FUNCTION_BLOCK FB_SiliconeProcess
VAR
    eState                  : E_SiliconeProcessState := E_SiliconeProcessState.Idle;
    bStartRequest           : BOOL;
    bStopRequest            : BOOL;
    bResetRequest           : BOOL;
    bReady                  : BOOL;
    bBusy                   : BOOL;
    bDone                   : BOOL;
    bFaulted                : BOOL;
	
	bVacuumBuildTimeoutFault   : BOOL;
	bVacuumLostFault           : BOOL;
	bVacuumReleaseTimeoutFault : BOOL;
	bEquipmentCompleteTimeoutFault : BOOL;

	
    bPinchValveRequest      : BOOL;
    bEquipmentStartRequest  : BOOL;
    bEquipmentStopRequest   : BOOL;
    bEquipmentResetRequest  : BOOL;
    stResult                : ST_ProcessResult;
    tonStep                 : TON;
	tSiliconeAirDelay 		: TIME;
END_VAR

// Runtime behaviour is implemented in Cyclic().

METHOD PUBLIC Cyclic
VAR_INPUT
    bSupplyReady               : BOOL;
    bEquipmentReady            : BOOL;
    bEquipmentBusy             : BOOL;
    bEquipmentDone             : BOOL;
    bEquipmentFaulted          : BOOL;
    stEquipmentResult          : ST_ProcessResult;
	bSiliconeStationPartPresent : BOOL;

    bSiliconeSupportExtended   : BOOL;
    bExtractorReady            : BOOL;
    bPartVacuumOk              : BOOL;
	tPartVacuumBuildTimeout    : TIME;
	tPartVacuumReleaseTimeout  : TIME;


    tPinchSettlingDelay        : TIME;
    tEquipmentStartTimeout     : TIME;
    tEquipmentCompleteTimeout  : TIME;
END_VAR

VAR_OUTPUT
    bPartVacuumEnable          : BOOL;
    bSiliconeAirEnable         : BOOL;
END_VAR
// Default one-scan handshake outputs.
bEquipmentStartRequest := FALSE;
bEquipmentStopRequest := FALSE;
bEquipmentResetRequest := FALSE;
bPartVacuumEnable := FALSE;
bSiliconeAirEnable := FALSE;

// Stop/reset are handled before state logic.
IF bResetRequest THEN
    bResetRequest := FALSE;
    bStartRequest := FALSE;
    bStopRequest := FALSE;
    bPinchValveRequest := FALSE;
    bPartVacuumEnable := FALSE;
	bSiliconeAirEnable := FALSE;
    bReady := bSupplyReady AND bEquipmentReady AND NOT bEquipmentFaulted;
    bBusy := FALSE;
    bDone := FALSE;
    bFaulted := FALSE;
	bVacuumBuildTimeoutFault := FALSE;
	bVacuumLostFault := FALSE;
	bVacuumReleaseTimeoutFault := FALSE;
	bEquipmentCompleteTimeoutFault := FALSE;
    stResult.bValid := FALSE;
    stResult.bPassed := FALSE;
    stResult.eCode := E_ProcessResultCode.None;
    stResult.udiFaultCode := 0;
    stResult.udiAlertCode := 0;
    stResult.usiRecipe := 0;
    bEquipmentResetRequest := TRUE;
    eState := E_SiliconeProcessState.Idle;
    tonStep(IN := FALSE);
    RETURN;
END_IF

IF bStopRequest THEN
    bStopRequest := FALSE;
    bStartRequest := FALSE;
    bPinchValveRequest := FALSE;
    bPartVacuumEnable := FALSE;
	bSiliconeAirEnable := FALSE;
    bBusy := FALSE;
    bDone := FALSE;
    bEquipmentStopRequest := TRUE;
    eState := E_SiliconeProcessState.Idle;
    tonStep(IN := FALSE);
    RETURN;
END_IF

// Any equipment fault while processing closes the flow path immediately.
IF bEquipmentFaulted
    AND (eState <> E_SiliconeProcessState.Idle)
    AND (eState <> E_SiliconeProcessState.Complete)
    AND (eState <> E_SiliconeProcessState.Fault)
THEN

    bPinchValveRequest := FALSE;
    bPartVacuumEnable := FALSE;
	bSiliconeAirEnable := FALSE;
    bBusy := FALSE;
    bDone := FALSE;
    bReady := FALSE;
    bFaulted := TRUE;

    stResult.bValid := FALSE;
    stResult.bPassed := FALSE;
    stResult.eCode := E_ProcessResultCode.EquipmentFault;

    eState := E_SiliconeProcessState.Fault;
END_IF

// Part holding vacuum must remain established while
// the silicone process is active.
IF NOT bPartVacuumOk
    AND (
        eState = E_SiliconeProcessState.WaitingAirBeforeSilicone
        OR eState = E_SiliconeProcessState.OpeningPinchValve
        OR eState = E_SiliconeProcessState.WaitingPinchSettling
        OR eState = E_SiliconeProcessState.StartingEquipment
        OR eState = E_SiliconeProcessState.WaitingEquipmentBusy
        OR eState = E_SiliconeProcessState.WaitingEquipmentComplete
        OR eState = E_SiliconeProcessState.ClosingPinchValve
        OR eState = E_SiliconeProcessState.WaitingAirAfterSilicone
    )
THEN

    bPinchValveRequest 			:= FALSE;
    bPartVacuumEnable 			:= FALSE;
	bSiliconeAirEnable 			:= FALSE;

    bEquipmentStartRequest 		:= FALSE;
    bEquipmentStopRequest 		:= TRUE;
	bVacuumLostFault 			:= TRUE;

    bReady 						:= FALSE;
    bBusy 						:= FALSE;
    bDone 						:= FALSE;
    bFaulted 					:= TRUE;
	stResult.bValid 			:= FALSE;
	stResult.bPassed 			:= FALSE;

    tonStep(IN := FALSE);
    eState 						:= E_SiliconeProcessState.Fault;

END_IF


CASE eState OF

    E_SiliconeProcessState.Idle:

        tonStep(IN := FALSE);

        bPinchValveRequest := FALSE;
        bPartVacuumEnable := FALSE;
		bSiliconeAirEnable := FALSE;
        bBusy := FALSE;
        bDone := FALSE;

        bReady :=
            bSupplyReady
            AND bEquipmentReady
            AND bSiliconeSupportExtended
            AND bExtractorReady
            AND NOT bEquipmentFaulted;

        IF bStartRequest AND bReady THEN
            bStartRequest := FALSE;
            bReady := FALSE;
            bBusy := TRUE;

            stResult.bValid := FALSE;
            stResult.bPassed := FALSE;

            eState := E_SiliconeProcessState.StartingVacuum;
        END_IF


   	E_SiliconeProcessState.StartingVacuum:

			bPinchValveRequest := FALSE;
			tonStep(IN := FALSE);
		
			// The part can only be detected after the Silicone Support is extended.
			// If no part is detected, finish the Silicone process as a valid FAIL.
			// Do not start the vacuum and do not run the IVEK.
			IF NOT bSiliconeStationPartPresent THEN
		
				bPartVacuumEnable := FALSE;
		
				bBusy := FALSE;
				bDone := TRUE;
				bReady := FALSE;
				bFaulted := FALSE;
		
				stResult.bValid := TRUE;
				stResult.bPassed := FALSE;
				stResult.eCode := E_ProcessResultCode.Fail;
		
				eState := E_SiliconeProcessState.Complete;
		
			ELSE
		
				bPartVacuumEnable := TRUE;
		
				eState := E_SiliconeProcessState.WaitingVacuumReady;
		
			END_IF
	
	
	E_SiliconeProcessState.WaitingVacuumReady:
	
		bPartVacuumEnable := TRUE;
		bPinchValveRequest := FALSE;
	
		tonStep(
			IN := TRUE,
			PT := tPartVacuumBuildTimeout
		);
	
		IF bPartVacuumOk THEN

			tonStep(IN := FALSE);
		
			eState := E_SiliconeProcessState.WaitingAirBeforeSilicone;
	
		ELSIF tonStep.Q THEN
	
			bPartVacuumEnable := FALSE;
			bPinchValveRequest := FALSE;
	
			bVacuumBuildTimeoutFault := TRUE;
			bFaulted := TRUE;
			bBusy := FALSE;
			bReady := FALSE;
			bDone := FALSE;
			
			stResult.bValid := FALSE;
			stResult.bPassed := FALSE;
	
			tonStep(IN := FALSE);
	
			eState := E_SiliconeProcessState.Fault;
	
		END_IF
		
		
	E_SiliconeProcessState.WaitingAirBeforeSilicone:

			bPartVacuumEnable := TRUE;
			bPinchValveRequest := FALSE;
			bSiliconeAirEnable := TRUE;
		
			tonStep(
				IN := TRUE,
				PT := tSiliconeAirDelay
			);
		
			IF tonStep.Q THEN
		
				tonStep(IN := FALSE);
		
				eState := E_SiliconeProcessState.OpeningPinchValve;
		
			END_IF
		
    E_SiliconeProcessState.OpeningPinchValve:

        bPartVacuumEnable := TRUE;
        bPinchValveRequest := TRUE;
		bSiliconeAirEnable := TRUE;

        tonStep(IN := FALSE);

        eState := E_SiliconeProcessState.WaitingPinchSettling;


    E_SiliconeProcessState.WaitingPinchSettling:

        bPartVacuumEnable := TRUE;
        bPinchValveRequest := TRUE;
		bSiliconeAirEnable := TRUE;

        tonStep(
            IN := TRUE,
            PT := tPinchSettlingDelay
        );

        IF tonStep.Q THEN
            tonStep(IN := FALSE);
            eState := E_SiliconeProcessState.StartingEquipment;
        END_IF


    E_SiliconeProcessState.StartingEquipment:

        bPartVacuumEnable := TRUE;
        bPinchValveRequest := TRUE;
		bSiliconeAirEnable := TRUE;

        IF bEquipmentReady THEN
            bEquipmentStartRequest := TRUE;

            tonStep(IN := FALSE);

            eState := E_SiliconeProcessState.WaitingEquipmentBusy;

        ELSE

            tonStep(
                IN := TRUE,
                PT := tEquipmentStartTimeout
            );

            IF tonStep.Q THEN
                bPinchValveRequest := FALSE;
                bPartVacuumEnable := FALSE;
				bSiliconeAirEnable := FALSE;
                bFaulted := TRUE;
                bBusy := FALSE;
				stResult.bValid := FALSE;
				stResult.bPassed := FALSE;

                eState := E_SiliconeProcessState.Fault;
            END_IF

        END_IF


    E_SiliconeProcessState.WaitingEquipmentBusy:

        bPartVacuumEnable := TRUE;
        bPinchValveRequest := TRUE;
		bSiliconeAirEnable := TRUE;

        // Keep Start asserted until the equipment acknowledges
        // the command by becoming Busy or Done.
        bEquipmentStartRequest := TRUE;

        tonStep(
            IN := TRUE,
            PT := tEquipmentStartTimeout
        );

        IF bEquipmentBusy OR bEquipmentDone THEN

            bEquipmentStartRequest := FALSE;

            tonStep(IN := FALSE);

            eState :=
                E_SiliconeProcessState.WaitingEquipmentComplete;

        ELSIF tonStep.Q THEN

            bEquipmentStartRequest := FALSE;
            bPinchValveRequest := FALSE;
            bPartVacuumEnable := FALSE;
			bSiliconeAirEnable := FALSE;
            bEquipmentStopRequest := TRUE;

            bFaulted := TRUE;
            bBusy := FALSE;
			stResult.bValid := FALSE;
			stResult.bPassed := FALSE;

            eState := E_SiliconeProcessState.Fault;

        END_IF


    E_SiliconeProcessState.WaitingEquipmentComplete:

        bPartVacuumEnable := TRUE;
        bPinchValveRequest := TRUE;
		bSiliconeAirEnable := TRUE;
		//bEquipmentCompleteTimeoutFault := TRUE;

        tonStep(
            IN := TRUE,
            PT := tEquipmentCompleteTimeout
        );

        IF bEquipmentDone THEN

            tonStep(IN := FALSE);
            eState := E_SiliconeProcessState.ClosingPinchValve;

        ELSIF tonStep.Q THEN

			bPinchValveRequest := FALSE;
			bPartVacuumEnable := FALSE;
			bSiliconeAirEnable := FALSE;
			bEquipmentStopRequest := TRUE;
		
			bEquipmentCompleteTimeoutFault := TRUE;
		
			bFaulted := TRUE;
			bBusy := FALSE;
		
			stResult.bValid := FALSE;
			stResult.bPassed := FALSE;
		
			eState := E_SiliconeProcessState.Fault;
		
		END_IF


    E_SiliconeProcessState.ClosingPinchValve:

			bPartVacuumEnable := TRUE;
			bSiliconeAirEnable := TRUE;
			bPinchValveRequest := FALSE;
	
			tonStep(IN := FALSE);
	
			eState := E_SiliconeProcessState.WaitingAirAfterSilicone;
			
			E_SiliconeProcessState.WaitingAirAfterSilicone:
	
		bPartVacuumEnable := TRUE;
		bPinchValveRequest := FALSE;
		bSiliconeAirEnable := TRUE;
	
		tonStep(
			IN := TRUE,
			PT := tSiliconeAirDelay
		);
	
		IF tonStep.Q THEN
	
			tonStep(IN := FALSE);
	
			eState := E_SiliconeProcessState.StoppingVacuum;
	
		END_IF


    E_SiliconeProcessState.StoppingVacuum:

        bPartVacuumEnable := FALSE;
        bPinchValveRequest := FALSE;

        tonStep(IN := FALSE);

        eState := E_SiliconeProcessState.WaitingVacuumReleased;


    E_SiliconeProcessState.WaitingVacuumReleased:

        bPartVacuumEnable := FALSE;
		bPinchValveRequest := FALSE;
		
		tonStep(
			IN := TRUE,
			PT := tPartVacuumReleaseTimeout
		);
		
		IF NOT bPartVacuumOk THEN
		
			tonStep(IN := FALSE);
		
			bBusy 				:= FALSE;
			bDone 				:= TRUE;
			bReady 				:= FALSE;
			
			stResult.bValid 	:= TRUE;
			stResult.bPassed 	:= TRUE;
			
			stResult.eCode 		:= E_ProcessResultCode.Pass;
			eState 				:= E_SiliconeProcessState.Complete;
		
		ELSIF tonStep.Q THEN
		
			bFaulted := TRUE;
			bBusy := FALSE;
			bReady := FALSE;
			bDone := FALSE;
			bVacuumReleaseTimeoutFault := TRUE;
			stResult.bValid := FALSE;
			stResult.bPassed := FALSE;
		
			tonStep(IN := FALSE);
		
			eState := E_SiliconeProcessState.Fault;
		
		END_IF

    E_SiliconeProcessState.Complete:

        bPartVacuumEnable := FALSE;
        bPinchValveRequest := FALSE;
		bSiliconeAirEnable := FALSE;
        bBusy := FALSE;
        bDone := TRUE;


    E_SiliconeProcessState.Fault:

        bPartVacuumEnable := FALSE;
        bPinchValveRequest := FALSE;
		bSiliconeAirEnable := FALSE;
        bReady := FALSE;
        bBusy := FALSE;
        bDone := FALSE;
        bFaulted := TRUE;

END_CASE
END_METHOD

METHOD PUBLIC GetEquipmentResetRequest : BOOL
VAR_INPUT
END_VAR
GetEquipmentResetRequest := bEquipmentResetRequest;
END_METHOD

METHOD PUBLIC GetEquipmentStartRequest : BOOL
VAR_INPUT
END_VAR
GetEquipmentStartRequest := bEquipmentStartRequest;
END_METHOD

METHOD PUBLIC GetEquipmentStopRequest : BOOL
VAR_INPUT
END_VAR
GetEquipmentStopRequest := bEquipmentStopRequest;
END_METHOD

METHOD PUBLIC GetPinchValveRequest : BOOL
VAR_INPUT
END_VAR
GetPinchValveRequest := bPinchValveRequest;
END_METHOD

METHOD PUBLIC GetResult : ST_ProcessResult
VAR_INPUT
END_VAR
GetResult := stResult;
END_METHOD

METHOD PUBLIC GetState : E_SiliconeProcessState
VAR_INPUT
END_VAR
GetState := eState;
END_METHOD

METHOD PUBLIC IsBusy : BOOL
VAR_INPUT
END_VAR
IsBusy := bBusy;
END_METHOD

METHOD PUBLIC IsDone : BOOL
VAR_INPUT
END_VAR
IsDone := bDone;
END_METHOD

METHOD PUBLIC IsFaulted : BOOL
VAR_INPUT
END_VAR
IsFaulted := bFaulted;
END_METHOD

METHOD PUBLIC IsReady : BOOL
VAR_INPUT
END_VAR
IsReady := bReady;
END_METHOD

METHOD PUBLIC RequestReset
VAR_INPUT
END_VAR
bResetRequest := TRUE;
END_METHOD

METHOD PUBLIC RequestStart
VAR_INPUT
END_VAR
IF bReady AND NOT bBusy AND NOT bFaulted THEN
    bStartRequest := TRUE;
END_IF
END_METHOD

METHOD PUBLIC RequestStop
VAR_INPUT
END_VAR
IF bBusy THEN bStopRequest := TRUE; END_IF
END_METHOD

END_FUNCTION_BLOCK

(* stored: Version 1.1.0.1, ProductVersion 3.1.4026.18
   POU FB_SiliconeProcess: Id {212587cd-c257-43af-acfd-e45649e0374c}, SpecialFunc None
   Method Cyclic: Id {b7a0fddb-671e-4115-a6a8-86f8d3cd3549}
   Method GetEquipmentResetRequest: Id {a5f7e317-f2a4-4c10-a4f0-228b42f92744}
   Method GetEquipmentStartRequest: Id {f6206d4d-f63c-425f-8808-7b0f6882fb28}
   Method GetEquipmentStopRequest: Id {c791fe21-9a54-4591-a1b8-c9ae5c5aabfa}
   Method GetPinchValveRequest: Id {e17faf55-b9a5-4402-8a52-3a087ef238a4}
   Method GetResult: Id {dc3638f4-5d08-4915-846a-68e0ad743f8b}
   Method GetState: Id {956ede30-ee9e-419c-9d1a-203ca3c81d00}
   Method IsBusy: Id {53fabbf5-919e-4dda-bce6-0e4c0320d6c9}
   Method IsDone: Id {f3c14b96-6269-44c5-9fea-1ca2d74f6607}
   Method IsFaulted: Id {75a6bcfc-9761-4be2-89c3-5116a3c844a3}
   Method IsReady: Id {fd56d7a3-a92b-4c53-8050-aead90e2b776}
   Method RequestReset: Id {c43f36b0-54e5-4f97-a3a9-f14919e999a3}
   Method RequestStart: Id {86b9333a-e110-4fa8-8e2e-b5391f88a843}
   Method RequestStop: Id {ff71cc52-5b6d-498f-93e3-65eeb616ec15} *)
